TYPE ID :
STRUCT
	intIndex			:	INT;
	sName				:	STRING;
	intMasterIndex		:	INT;
END_STRUCT
END_TYPE

(* stored: Version 1.1.0.1, ProductVersion 3.1.4024.6
   DUT ID: Id {7d14d8b8-cf28-48fe-98b4-993958eeac33} *)
